FUNCTION_BLOCK CL_AxisL1LeftBack EXTENDS CL_AxisRobot
var
END_VAR

SUPER^();

METHOD PROTECTED InitDefect : BOOL
sWhichAxis := 'left(L1)-back';
InitDefect := true;
END_METHOD

METHOD PROTECTED InitParams : BOOL
VAR_INPUT
END_VAR
InitParams := super^.InitParams();
_lrInverse := 1.0;
END_METHOD

END_FUNCTION_BLOCK

(* stored: Version 1.1.0.1, ProductVersion 3.1.4024.12
   POU CL_AxisL1LeftBack: Id {471b1620-a4eb-4e45-adf5-d1968ea43216}, SpecialFunc None
   Method InitDefect: Id {eae795de-6055-4462-8fdf-b6c77b3c5095}
   Method InitParams: Id {fde22834-ed60-4fc7-bb5f-c3c336426d56} *)
